{attribute 'qualified_only'}
{attribute 'strict'}
{attribute 'to_string'}
TYPE E_STATION_TYPE :
(
	INVALID,
  STATION_PROCESS,      // default station with/without process
  STATION_GEAR_IN_POS   // GearInPos station for flying saw with MasterAxis
)USINT;
END_TYPE

(* stored: Version 1.1.0.1, ProductVersion 3.1.4026.20
   DUT E_STATION_TYPE: Id {b9c4dfbd-9b9d-41e4-bcb0-2befb5c7907e} *)
